{attribute 'qualified_only'}
{attribute 'strict'}
{attribute 'to_string'}
TYPE eTcaWorkpiecePlaceProgress :
(
	undefined := 0,
	blank,
	inProcess,
	finished,
	Error,
	
	MAXSIZE
);
END_TYPE

(* stored: Version 1.1.0.1
   DUT eTcaWorkpiecePlaceProgress: Id {85a7e9b2-9e2f-4e38-b696-1020260b8304} *)
